Yaskawa INFORM job: R1_W66-W67(-70,-90)KM-OK.JBI

/JOB
//NAME R1_W66-W67(-70,-90)KM-OK
///FOLDERNAME KRIS-SCIANA
//POS
///NPOS 39,39,0,3,0,0
///TOOL 0
///POSTYPE PULSE
///PULSE
C00000=-135635,-24500,-41716,31750,82638,33791
C00001=-121173,28136,37388,9783,95382,11090
C00002=-121152,31888,45574,9734,92313,10856
C00003=-121142,35145,50794,9721,90794,10743
C00004=-121143,35483,52754,9718,89774,10663
C00005=-121143,35225,52204,9718,89977,10679
C00006=-121140,38719,56440,9718,89178,10618
C00007=-121176,37573,54181,9710,89973,10668
C00008=-120187,34889,50757,9920,90573,11044
C00009=-119360,34923,50783,10093,90475,11313
C00010=-120187,34889,50757,9920,90573,11044
C00011=-120195,33129,47147,9931,91873,11144
C00012=-120213,29283,38831,9979,94971,11386
C00013=-124262,41791,46564,-15679,81195,12986
C00014=-125301,47706,56682,-15822,77923,13043
C00015=-124319,51586,62900,-15917,76347,13598
C00016=-124340,50707,62802,-15941,75964,13642
C00017=-124340,50450,62252,-15928,76164,13616
C00018=-124303,54143,66935,-15991,75223,13754
C00019=-124340,48208,57292,-15821,77994,13376
C00020=-118829,36803,52428,-28844,69518,21730
C00021=-119649,36749,52382,-28805,69244,21478
C00022=-118829,36803,52428,-28844,69518,21730
C00023=-118147,34363,48669,-28702,70681,21695
C00024=-116410,28824,40027,-28425,73448,21667
C00025=-120722,36277,52307,21922,60833,-8108
C00026=-120725,29599,36610,20842,66654,-6972
C00027=-109986,44671,45472,4739,72285,39309
C00028=-109829,25936,29329,1019,58563,75027
C00029=-109240,33530,46226,1186,52861,75214
C00030=-120730,33890,48639,21720,61795,-7914
C00031=-120725,33272,48739,21793,61440,-7984
C00032=-141146,38851,52736,5146,51589,62144
C00033=-136543,33769,49960,-8490,46897,65257
C00034=-136074,16665,19493,-866,53899,64440
C00035=-141194,19904,22517,1630,53727,62321
C00036=-132020,10447,-13346,-2437,70990,65718
C00037=-130510,-84668,-101602,-2499,71155,65752
C00038=-130510,-84668,-101602,-2499,71155,65752
BC00000=108096,720728,946792
BC00001=156025,809067,742793
BC00002=156025,809067,742793
BC00003=156025,809067,742793
BC00004=156025,809067,742793
BC00005=156025,809067,742793
BC00006=156025,809067,742793
BC00007=156025,809067,742793
BC00008=156025,809067,742793
BC00009=156025,809067,742793
BC00010=156025,809067,742793
BC00011=156025,809067,742793
BC00012=156025,809067,742793
BC00013=112859,763833,697825
BC00014=112859,763833,697825
BC00015=112859,763833,697825
BC00016=112859,763833,697825
BC00017=112859,763833,697825
BC00018=112859,763833,697825
BC00019=112859,763833,697825
BC00020=112859,763833,697825
BC00021=112859,763833,697825
BC00022=112859,763833,697825
BC00023=112859,763833,697825
BC00024=112859,763833,697825
BC00025=130925,744955,838542
BC00026=131347,744951,731016
BC00027=135195,751313,703596
BC00028=135195,751313,703596
BC00029=135195,751313,703596
BC00030=135195,751313,703596
BC00031=135195,751313,703596
BC00032=135194,751312,703593
BC00033=135194,751312,703593
BC00034=135194,751312,703593
BC00035=135194,751312,703593
BC00036=135194,751312,703593
BC00037=135194,751312,885398
BC00038=135194,686612,885398
///POSTYPE BASE
///RECTAN
///RCONF 0,0,0,0,0,0,0,0,0,0,0,0,0,0,0,0,0,0,0,0,0,0,0,0
P00006=0.222,-3.123,-1.508,0.0000,0.0000,0.0000
P00021=-0.225,-6.128,-0.405,0.0000,0.0000,0.0000
P00022=0.222,-3.123,-1.508,0.0000,0.0000,0.0000
//INST
///DATE 2024/07/23 15:55
///ATTR SC,RW
///GROUP1 RB1,BS1
NOP
'r2_W66-W67(-70,-90)
MOVJ C00000 BC00000 VJ=50.00
'Path S1112 (for W504)
SFTOF
MOVJ C00001 BC00001 VJ=80.00
MOVJ C00002 BC00002 VJ=100.00
MOVL C00003 BC00003 V=60.0
REFP 3 C00004 BC00004
CALL JOB:SEARCH-R1
SET P021 P006
SFTON P021
MOVL C00005 BC00005 V=60.0
REFP 3 C00006 BC00006
CALL JOB:SEARCH-R1
SET P021 P006
SFTON P021
MOVL C00007 BC00007 V=60.0
MOVL C00008 BC00008 V=60.0
REFP 3 C00009 BC00009
CALL JOB:SEARCH-R1
SET P021 P006
SFTON P021
MOVL C00010 BC00010 V=60.0
MOVL C00011 BC00011 V=100.0
MOVL C00012 BC00012 V=100.0
'Path S1113 (for W504)
SFTOF
MOVJ C00013 BC00013 VJ=100.00
MOVJ C00014 BC00014 VJ=100.00
MOVL C00015 BC00015 V=60.0
REFP 3 C00016 BC00016
CALL JOB:SEARCH-R1
SET P022 P006
SFTON P022
MOVL C00017 BC00017 V=60.0
REFP 3 C00018 BC00018
CALL JOB:SEARCH-R1
SET P022 P006
SFTON P022
MOVL C00019 BC00019 V=60.0
MOVL C00020 BC00020 V=60.0
REFP 3 C00021 BC00021
CALL JOB:SEARCH-R1
SET P022 P006
SFTON P022
MOVL C00022 BC00022 V=60.0
MOVL C00023 BC00023 V=100.0
MOVL C00024 BC00024 V=100.0
'Path W1114
SFTOF
SFTON P021
MOVJ C00025 BC00025 VJ=100.00
MOVJ C00026 BC00026 VJ=100.00
MOVJ C00027 BC00027 VJ=100.00
MOVJ C00028 BC00028 VJ=100.00
MOVL C00029 BC00029 V=100.0 PL=0
REFP 1 C00030 BC00030
REFP 2 C00031 BC00031
MACRO1 MJ#(0) ARGF7
ARCON
SFTOF
SFTON P022
MOVL C00032 BC00032 V=10.0
MOVL C00033 BC00033 V=10.0
ARCOF
MOVL C00034 BC00034 V=333.3
SFTOF
MOVL C00035 BC00035 V=333.3
MOVJ C00036 BC00036 VJ=100.00
MOVJ C00037 BC00037 VJ=100.00
MOVJ C00038 BC00038 VJ=100.00
END
